INTERFACE IOutputDevice EXTENDS IDevice

METHOD UpdateOutputsFromState
VAR_IN_OUT CONSTANT
	executionContext : AUTOMATION_EXECUTION_CONTEXT;
	aggregateException : Core.AggregateException;
END_VAR
END_METHOD

END_INTERFACE

(* stored: Version 1.1.0.1
   Itf IOutputDevice: Id {9ff1eac2-7c3a-4e18-b5c3-83d36d605c6c}
   Method UpdateOutputsFromState: Id {5eb289e0-048e-4fb1-b4b5-450d3a21a673} *)
